PROGRAM OP10_SCN_ENB
VAR
END_VAR

END_PROGRAM

(* stored: Version 1.1.0.1, ProductVersion 3.1.4024.11
   POU OP10_SCN_ENB: Id {49e8c792-f153-4236-b50d-2ccc42448579}, SpecialFunc None *)
